TYPE TimedPulse :
STRUCT
	tLeadingGap: TIME   := T#0MS;
	tHighSignal: TIME := T#0MS;
	tTrailingGap: TIME:= T#0MS;
END_STRUCT
END_TYPE

(* stored: Version 1.1.0.1, ProductVersion 3.1.4024.15
   DUT TimedPulse: Id {1cf71819-5efd-4778-9318-886e6b804f24} *)
